FUNCTION_BLOCK FB_ToggleButton
VAR_INPUT
	bIsToggleButtonOn : BOOL;
END_VAR
VAR_OUTPUT
	bLightOfToggleButton : BOOL;
END_VAR
VAR
	fbToggle_RTRIG : R_TRIG;
END_VAR

// When a button is clicked, turn light on if it was off, or turn light off if it was on
fbToggle_RTRIG(clk := bIsToggleButtonOn);
IF fbToggle_RTRIG.Q THEN
	bLightOfToggleButton := NOT bLightOfToggleButton;
END_IF

END_FUNCTION_BLOCK

(* stored: Version 1.1.0.1, ProductVersion 3.1.4024.12
   POU FB_ToggleButton: Id {01df59ea-0cbb-471a-9285-fb67bdce7be4}, SpecialFunc None *)
